// TIA Portal V19 export
VAR_GLOBAL   // PLC tag table "LB211"
   LB211_DeadMan_Ch1 AT %I1079.0 : Bool;   // 106DI0 - 234SB1
   LB211_DeadMan_Ch2 AT %I1079.4 : Bool;   // 106DI4 - 234SB1
   LB211_Pb_Minus AT %I123.3 : Bool;   // 336SB1
   LB211_Pb_Plus AT %I123.4 : Bool;   // 336SB2
END_VAR
